// TIA Portal V19 export
FUNCTION "FlyingCarriage_CALL" : Void   // FC160, LAD
// stored: SetENOAutomatically false
   VAR_TEMP
      MissIO : Bool;
   END_VAR
BEGIN

REGION Network 1: Data In - PB
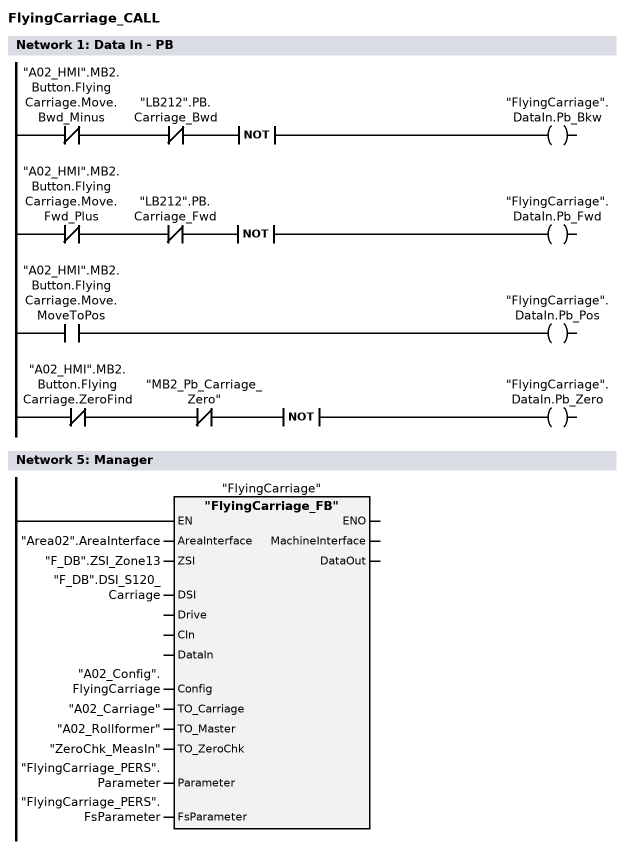
   RUNG wire#powerrail
      I_Contact( "A02_HMI".MB2.Button.FlyingCarriage.Move.Bwd_Minus )
      I_Contact( "LB212".PB.Carriage_Bwd )
      Not()
      Coil( "FlyingCarriage".DataIn.Pb_Bkw )
   END_RUNG
   RUNG wire#powerrail
      I_Contact( "A02_HMI".MB2.Button.FlyingCarriage.Move.Fwd_Plus )
      I_Contact( "LB212".PB.Carriage_Fwd )
      Not()
      Coil( "FlyingCarriage".DataIn.Pb_Fwd )
   END_RUNG
   RUNG wire#powerrail
      Contact( "A02_HMI".MB2.Button.FlyingCarriage.Move.MoveToPos )
      Coil( "FlyingCarriage".DataIn.Pb_Pos )
   END_RUNG
   RUNG wire#powerrail
      I_Contact( "A02_HMI".MB2.Button.FlyingCarriage.ZeroFind )
      I_Contact( "MB2_Pb_Carriage_Zero" )
      Not()
      Coil( "FlyingCarriage".DataIn.Pb_Zero )
   END_RUNG
   // the same network as SCL:
   "FlyingCarriage".DataIn.Pb_Bkw := NOT (NOT "A02_HMI".MB2.Button.FlyingCarriage.Move.Bwd_Minus AND NOT "LB212".PB.Carriage_Bwd);
   "FlyingCarriage".DataIn.Pb_Fwd := NOT (NOT "A02_HMI".MB2.Button.FlyingCarriage.Move.Fwd_Plus AND NOT "LB212".PB.Carriage_Fwd);
   "FlyingCarriage".DataIn.Pb_Pos := "A02_HMI".MB2.Button.FlyingCarriage.Move.MoveToPos;
   "FlyingCarriage".DataIn.Pb_Zero := NOT (NOT "A02_HMI".MB2.Button.FlyingCarriage.ZeroFind AND NOT "MB2_Pb_Carriage_Zero");
END_REGION

REGION Network 2 (SCL): Data In - Sensor

   "FlyingCarriage".DataIn.Fbk_Fan := FALSE;
END_REGION

REGION Network 3 (SCL): Drive

   "FlyingCarriage".Drive.Infeed_ON := "Areas_ITF".AG.Infeed_Running;
   "FlyingCarriage".Drive.AccessPoint := "HW_Const_Values".CU2_PN_585A1_ModuleAccessPoint;
   "FlyingCarriage".Drive.AxisID := "CU2_ID_3_1300A1_1300M1";
   "FlyingCarriage".Drive.TokenChain := "TOKENCHAIN_CU2";
END_REGION

REGION Network 4 (SCL): Cin
   "FlyingCarriage".CIn := "RollformingMng".COut.FlyingCarriage;

   "FlyingCarriage".CIn.ToolAtRest := "FinalCut".COut.AllAtRest;
   "FlyingCarriage".CIn.ToolAtRestManEmptyng := "FinalCut".COut.CutHead.Rest AND "FinalCut".COut.MarkHead.Rest;
END_REGION

REGION Network 5: Manager
   RUNG wire#powerrail
      "FlyingCarriage"(AreaInterface := "Area02".AreaInterface, ZSI := "F_DB".ZSI_Zone13, DSI := "F_DB".DSI_S120_Carriage, Drive :=, CIn :=, DataIn :=, Config := "A02_Config".FlyingCarriage, TO_Carriage := "A02_Carriage", TO_Master := "A02_Rollformer", TO_ZeroChk := "ZeroChk_MeasIn", Parameter := "FlyingCarriage_PERS".Parameter, FsParameter := "FlyingCarriage_PERS".FsParameter, MachineInterface =>, DataOut =>)
   END_RUNG
   // the same network as SCL:
   "FlyingCarriage"(AreaInterface := "Area02".AreaInterface,   // "FlyingCarriage_FB"
                    ZSI := "F_DB".ZSI_Zone13,
                    DSI := "F_DB".DSI_S120_Carriage,
                    Config := "A02_Config".FlyingCarriage,
                    TO_Carriage := "A02_Carriage",
                    TO_Master := "A02_Rollformer",
                    TO_ZeroChk := "ZeroChk_MeasIn",
                    Parameter := "FlyingCarriage_PERS".Parameter,
                    FsParameter := "FlyingCarriage_PERS".FsParameter);
END_REGION

REGION Network 6 (SCL): Data Out
   "MB2_Lp_Carriage_Zero" := "FlyingCarriage".DataOut.LP_ZeroOK;
END_REGION
END_FUNCTION
